// TIA Portal V19 export
VAR_GLOBAL   // PLC tag table "Equipment_Template_12"
END_VAR
